{attribute 'linkalways'} 
{attribute 'no_explicit_call' := 'This FB is a CLASS and must be accessed using methods or properties'}
{attribute 'enable_dynamic_creation'}
FUNCTION_BLOCK _ULINT EXTENDS IntegerDatatypeBase
VAR
	localData : ULINT;
	activeData : REFERENCE TO ULINT REF= localData;
END_VAR

PROPERTY PUBLIC Address : PVOID
GET
Address := ADR(activeData);
END_GET
END_PROPERTY

METHOD PUBLIC ClearReference
VAR_INPUT
END_VAR
activeData REF= localData;
END_METHOD

METHOD PUBLIC Clone : I_Datatype
VAR
    pClone : POINTER TO _ULINT;
END_VAR
pClone := __NEW(_ULINT(InitialValue := Value));
Clone := pClone^;
END_METHOD

PROPERTY PUBLIC Datatype : T_MAXSTRING
GET
Datatype := 'ULINT';
END_GET
END_PROPERTY

METHOD FB_init : BOOL
VAR_INPUT
	bInitRetains : BOOL; // if TRUE, the retain variables are initialized (warm start / cold start)
	bInCopyCode : BOOL;  // if TRUE, the instance afterwards gets moved into the copy code (online change)
	InitialValue : ULINT;
END_VAR
localData := InitialValue;
END_METHOD

PROPERTY PUBLIC IsSigned : BOOL
GET
IsSigned := FALSE;
END_GET
END_PROPERTY

PROPERTY PUBLIC LowerBound : ULINT
GET
LowerBound := DatatypeLimits.ULINT_LOWER_LIMIT;
END_GET
END_PROPERTY

METHOD PUBLIC MakeReferenceTo
VAR_INPUT
	ReferenceTarget : REFERENCE TO ULINT;
END_VAR
activeData REF= ReferenceTarget;
END_METHOD

METHOD PROTECTED SerializeLowerbound
VAR_INPUT
	Serializer : I_Serializer;
END_VAR
Serializer.AddLint(Lowerbound);
END_METHOD

METHOD PROTECTED SerializeUpperbound
VAR_INPUT
	Serializer : I_Serializer;
END_VAR
Serializer.AddLint(Upperbound);
END_METHOD

METHOD PUBLIC SerializeWith
VAR_INPUT
	Serializer : I_Serializer;
END_VAR
Serializer.AddUlint(activeData);
END_METHOD

PROPERTY PUBLIC Size : UDINT
GET
Size := SIZEOF(activeData);
END_GET
END_PROPERTY

METHOD TryDeserializeFrom : BOOL
VAR_INPUT
	Deserializer : I_Deserializer;
	Feedback : I_DeserializerFeedback;
END_VAR
TryDeserializeFrom := Deserializer.TryGetUlint(activeData, Feedback);
END_METHOD

METHOD TryMakeReferenceTo : BOOL
VAR_INPUT
	Target : I_Datatype;
END_VAR
VAR
	pTargetData : POINTER TO ULINT;
END_VAR
IF NOT (Target.Datatype = Datatype) THEN
	RETURN;
END_IF

pTargetData := Target.Address;
activeData REF= pTargetData^;
TryMakeReferenceTo := TRUE;
END_METHOD

PROPERTY PUBLIC UpperBound : ULINT
GET
UpperBound :=  DatatypeLimits.ULINT_UPPER_LIMIT;
END_GET
END_PROPERTY

PROPERTY PUBLIC Value : ULINT
GET
Value := activeData;
END_GET
SET
activeData := Value;
END_SET
END_PROPERTY

END_FUNCTION_BLOCK

(* stored: Version 1.1.0.1, ProductVersion 3.1.4024.12
   POU _ULINT: Id {c7898852-3f8c-06ea-37d8-fdb1eefce63a}, SpecialFunc None
   Folder Constructor: Id {c056bdcf-aa40-02f2-177e-270978828ede}
   Folder Protected: Id {e31aa3f5-6766-075e-3ec1-51cdaa3906b9}
   Property Address: Id {e633fbea-6deb-07a1-0f6b-d3d8dd5ece97}
   Get Get: Id {afe0d9d2-7d19-05aa-0752-b3b7e2c677da}
   Method ClearReference: Id {29033a30-bfed-0588-36c1-d883e0c55df2}
   Method Clone: Id {7904eb54-5a5e-0db0-0d3d-2dba99f8e7c1}
   Property Datatype: Id {47bd40c2-540b-0011-12d3-a3542e29e63d}
   Get Get: Id {f24b824f-7f93-056a-3ca6-5b9baea73d1c}
   Method FB_init: Id {c56a88d2-c768-0b03-1c92-8f5cec67c152}
   Property IsSigned: Id {75e0dece-c871-0ada-03d1-569478bc9ae6}
   Get Get: Id {b72acb2c-9416-0074-0851-ec8dd8cb543c}
   Property LowerBound: Id {2b5124b7-c4b8-07a2-01ee-2bbc83277354}
   Get Get: Id {e2455522-3265-0484-03f2-f2715c53694d}
   Method MakeReferenceTo: Id {27b89260-d794-0105-263d-7c750ae1e15f}
   Method SerializeLowerbound: Id {06666c40-7115-0593-257e-7ea5cb9c8d05}
   Method SerializeUpperbound: Id {43843877-346d-0ebd-34a6-ec5ecb7f5c6f}
   Method SerializeWith: Id {6efedb8d-ee30-00ea-0b6d-8e64df3fd52f}
   Property Size: Id {f7802e2e-e844-04b3-278f-6b3a96c74472}
   Get Get: Id {135cfe1d-99e7-0c73-3f30-fa288c706f6a}
   Method TryDeserializeFrom: Id {0b0ad417-a689-0263-08b8-8a3b54693546}
   Method TryMakeReferenceTo: Id {1ba40e25-354a-054d-2471-d4811c1c7d48}
   Property UpperBound: Id {377ba917-fc59-0030-293a-70175826ab29}
   Get Get: Id {27ef2049-0590-0dfc-2ed3-19751e227321}
   Property Value: Id {4dda2ae8-674a-0fb8-2bf8-7e756f7ae32e}
   Get Get: Id {c8a59718-4109-0b1f-2727-4c90670fc004}
   Set Set: Id {d99615b2-e08b-04bb-2005-0a910135f29c} *)
